PROGRAM FC1
VAR
END_VAR

END_PROGRAM

(* stored: Version 1.1.0.1, ProductVersion 3.1.4022.12
   POU FC1: Id {937363ea-ad41-4b81-afaf-d5c68b6c65ee}, SpecialFunc None *)
